PROGRAM MAIN
VAR
	//Control mode
	eMode : E_ControlMode := E_ControlMode.Auto;
	
	// Heat supply circle
	fbHSS		: FB_HSS;

	//simulated sensor data
	fbHSSSenDa	: FB_SenDaHydMixCir;
	//simulated enviromental temperature
	fbAmbientAir : FB_AmbientAir;		
								 
END_VAR

//Check main control mode
eMode := ADS.eModeMainControlModeADS;
//Set control modes
IF eMode = E_ControlMode.ExternalADSControl THEN		
	fbHSS.Mode 	:= ADS.eModeHSSADS;	
ELSE	
	fbHSS.Mode 	:= eMode;
END_IF

//Simulated the sensor tmeprature and enviromental temperature
 
fbHSSSenDa.Run();
fbAmbientAir.Run();

//Raw temperature input 
fbHSS.TempSupPrim := fbHSSSenDa.fTempSupPrimAct;
fbHSS.TempRetPrim := fbHSSSenDa.fTempRetPrimAct;
fbHSS.TempRet := fbHSSSenDa.fTempRetAct;
fbHSS.TempSup := fbHSSSenDa.fTempSupAct;
//Valve input
fbHSS.Valve := fbHSSSenDa.fHSSValveAct;


//Execute Routine 
fbHSS.Run();

END_PROGRAM

(* stored: Version 1.1.0.1, ProductVersion 3.1.4024.6
   POU MAIN: Id {739250fd-a178-4b07-8586-e950252efe80}, SpecialFunc None *)
